// TwinCAT 3 PLC project Washing_Machine_Simulator
// ProgramVersion: 3.1.4024.0
// libraries:
//   Tc2_Standard, * (Beckhoff Automation GmbH)
//   Tc2_System, * (Beckhoff Automation GmbH)
//   Tc3_Module, * (Beckhoff Automation GmbH)
// project tree:
//   DUTs/ E_StateType.TcDUT, E_StrategyType.TcDUT
//   / PlcTask.TcTTO
//   POUs/ FB_HeavyWash.TcPOU (not stored), FB_NormalWash.TcPOU (not stored), FB_SoftWash.TcPOU (not stored), FB_WashingMachine.TcPOU (not stored), I_WashStrategy.TcIO (not stored), MAIN.TcPOU (not stored)
// real-time tasks:
//   TASK PlcTask: cycle T#10ms, priority 20, ADS port 350

CONFIGURATION Washing_Machine_Simulator
    RESOURCE PLC ON TwinCAT3
        TASK PlcTask(INTERVAL := T#10ms, PRIORITY := 20);
        PROGRAM MAIN WITH PlcTask : MAIN;
    END_RESOURCE
END_CONFIGURATION

// ---- DUTs/E_StateType.TcDUT
{attribute 'qualified_only'}
{attribute 'strict'}
TYPE E_StateType :
(
	Idle,
	Filling,
	Washing,
	Draining,
	Rinse,
	Completed
);
END_TYPE

// ---- DUTs/E_StrategyType.TcDUT
{attribute 'qualified_only'}
{attribute 'strict'}
TYPE E_StrategyType :
(
	HeavyWash,
	NormalWash,
	SoftWash,
	None
);
END_TYPE
